(* IEC 61131-3 sources: HPLC/template/projeto-plc/globals, 5 files *)

(* ---- 00_GVL_IO.st ---- *)
VAR_GLOBAL
    InputsDigitais : ST_EntradasDigitais;
    InputsAnalogicos : ST_EntradasAnalogicas;
    OutputsDigitais : ST_SaidasDigitais;
    HabilitaSimulacao : BOOL := TRUE;
END_VAR

(* ---- 10_GVL_PROCESSO.st ---- *)
VAR_GLOBAL
    PressaoJusante : ST_InstrumentoAnalogico;
    TemperaturaOleo : ST_InstrumentoAnalogico;
    PIT700 : ST_InstrumentoAnalogico;
    PIT701 : ST_InstrumentoAnalogico;
    PIT702 : ST_InstrumentoAnalogico;
    PIT703 : ST_InstrumentoAnalogico;
    PIT704 : ST_InstrumentoAnalogico;
    PIT705 : ST_InstrumentoAnalogico;
    TIT700 : ST_InstrumentoAnalogico;
    TIT701 : ST_InstrumentoAnalogico;
    TIT702 : ST_InstrumentoAnalogico;
    TIT703 : ST_InstrumentoAnalogico;
    TIT704 : ST_InstrumentoAnalogico;
    MotorPrincipal : ST_Motor;
    MotorExaustor : ST_Motor;
    MotorVentilador1 : ST_Motor;
    MotorVentilador2 : ST_Motor;
    ValvulaSucao : ST_Valvula;
END_VAR

(* ---- 20_GVL_CONTROLE.st ---- *)
VAR_GLOBAL
    Comandos : ST_Comandos;
    ComandoConsolidado : ST_ComandoConsolidado;
    StatusMaquina : ST_StatusMaquina;
    SetpointCarga : REAL := 5.5;
    SetpointAlivio : REAL := 8.0;
    (* Simulação rápida: cada transição pode ocorrer no próximo scan de 10 ms. *)
    TempoMinimoEstado : TIME := T#0ms;
END_VAR

(* ---- 30_GVL_SUPERVISAO.st ---- *)
VAR_GLOBAL
    IHMEstadoAtual : INT;
    IHMPressao : REAL;
    IHMTemperatura : REAL;
    IHMPronto : BOOL;
    IHMEmOperacao : BOOL;
    IHMEmFalha : BOOL;
    TotalTrips : UDINT;
END_VAR

(* ---- 40_GVL_RETENTIVOS.st ---- *)
VAR_GLOBAL
    TotalPartidas : UDINT;
    HorimetroCargaSegundos : UDINT;
    HorimetroAlivioSegundos : UDINT;
    SolicitaResetFabrica : BOOL;
    SolicitaAtualizaFabrica : BOOL;
END_VAR
